// TIA Portal V19 export
ORGANIZATION_BLOCK "A02_OB30"   // OB30, LAD, CyclicInterrupt
// stored: SetENOAutomatically false
   VAR_INPUT
      Initial_Call : Bool;   // Initial call of this OB
      Event_Count : Int;   // Events discarded
   END_VAR
BEGIN

REGION Network 1
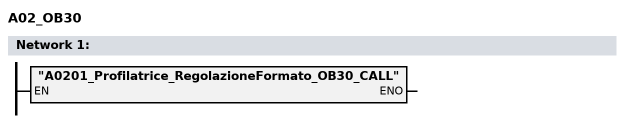
   RUNG wire#powerrail
      "A0201_Profilatrice_RegolazioneFormato_OB30_CALL"()
   END_RUNG
   // the same network as SCL:
   "A0201_Profilatrice_RegolazioneFormato_OB30_CALL"();
END_REGION
END_ORGANIZATION_BLOCK
